// TIA Portal V19 export
VAR_GLOBAL   // PLC tag table "Entrées"
   PART_AV AT %I0.0 : Bool;   // Détection pièce disponible
   B2 AT %I0.1 : Bool;   // Détection pièces (pas noir)
   B4 AT %I0.2 : Bool;   // Barrière sécurité
   "1B1" AT %I0.4 : Bool;   // Vérin 1A1 position haute
   "1B2" AT %I0.5 : Bool;   // Vérin 1A1 position basse
   "2B1" AT %I0.6 : Bool;   // Vérin 2A1 rentré
   Start AT %I1.0 : Bool;   // Départ cycle
   Stop AT %I1.1 : Bool;   // Fin cycle
   Reset AT %I1.3 : Bool;   // Initialisation station
   Analogique AT %IW800 : Int;   // Capteur analogique
END_VAR
